Staubli VAL3: _remote.pgx

program _remote()
  local bool bActive
  local InstrItem l_iProg
  local string message
  local string sString
begin
  bActive=false
  switch nRemoteID
    case 0
      // START
      if taskStatus("Cycle")==-1
        logMsg("[KERNEL] SUPERVISOR:REMOTE>Start cycle")
        cycleStatus:bToStart=true
      endIf
      bActive=true
    break
    case 1
      //STOP
      cycleStatus:bToStop=true
      bActive=true
    break
    case 2
      //END CYCLE
      if taskStatus("Cycle")!=-1
        logMsg("[KERNEL] SUPERVISOR:REMOTE>End cycle")
        cycleStatus:bToEnd=true
      endIf
      bActive=true
    break
    case 3
      // HOME STRATEGY
      if taskStatus("Cycle")==-1
        logMsg("[KERNEL] SUPERVISOR:REMOTE>Home strategy")
        cycleStatus:bToHome=true
      endIf
      bActive=true
    break
    case 4
      // simulation of the program
      l_iProg.sType="PROG"
      l_iProg.sData=sRemoteID
      call _startSimul(l_iProg)
      logMsg("[KERNEL] SUPERVISOR:REMOTE>insert the program: "+sRemoteID)
      bActive=true
    break
  endSwitch
  if bActive
    nRemoteID=-1
    sRemoteID=""
    if taskStatus("Interface")==0
      taskResume("Interface",0)
    endIf
  endIf
end
